// TIA Portal V19 export
DATA_BLOCK "DB_DP"   // DB85
{ S7_Optimized_Access := 'FALSE' }
// stored: AutoNumber false
   VAR RETAIN
      Anz_DP : Int := 2;   // * Anzahl Dosierpumpen
      Offset : Int := 20;   // * Beginn Daten
      leng_Pos : Int := 20;   // * Länge Daten
      DP_Nr : Int := 0;   // Nummer der aktuell bearbeiteten Pumpe
      Sekunden_Takt : Bool := FALSE;   // merkt sich den Sekundentakt
      Minuten_Takt : Bool := FALSE;   // eine Minute ist um (für einen Umlauf an)
      HandeventTakt : Bool := FALSE;   // zyklischer Abstand Meldung manuelle Zugabe
      res1 : Bool := FALSE;
      res2 : Bool := FALSE;
      res3 : Bool := FALSE;
      res4 : Bool := FALSE;
      res5 : Bool := FALSE;
      AM_Minute : Byte := 16#32;   // Altmerker Minute
      MinCount : Int := 1;   // Minutenzähler (10min)
      CheckPU : Int := 0;   // Kontrollpumpe
      resI : Int := 0;
      resD1 : DWord := 16#0000_0000;
      DP : Array[0..20] of Struct   // * Feldlänge anpassen
         Typ : Byte;   // *VAT 0=Menge Zeit,1=Menge Pulse,2=Handzugabe,5=H2O
         LaZa_Nr : Byte;   // *VAT Ladungszähler-Nr.
         EventTime : Int;   // 0=jede Dosierung sonst Zeit in Minuten
         Rest_EventTime : Int;   // Restzeit bis nächstes Event
         DP_Start : Bool;   // Start Dosierpumpe (auch extern 1 Autowert)
         DP_OFF : Bool;   // ext.Abschaltg. zB.Motorschutz oä.
         DP_Hand : Bool;   // Start eine Handzugabe
         DP_Strg : Bool;   // Störung Dosierpumpe
         DP_Imp : Bool;   // externer Zählimpuls
         DP_Niv : Bool;   // Niveau max erreicht
         DP_IN6 : Bool;
         DP_IN7 : Bool;
         DP_IN8 : Bool;
         Dosi_akt : Bool;   // Nachdosierung aktiv
         AM_Dosi : Bool;   // Altmerker Dosierung
         Meldung : Bool;   // Dosierung melden
         AM_Strg : Bool;   // Altmerker Störung
         DP_ext_Imp : Bool;   // Pumpe wird extern betrieben (Impuls wird als Eingang geliefert)
         res4 : Bool;
         AM_DP_Start : Bool;   // Merker DP Start
         RestZeit : Int;   // Restzeit Zähler Dosierimpuls/Pausenzeit
         DosMenge_Auto : Real;   // Dosiermenge Automatik
         DosMenge_Hand : Real;   // Dosiermenge Handzugabe
         ZeitBasis : Byte;   // Zeitbasis für Kalibrierung 0=s 1=min 2=h
         Korr_Einheit : Byte;   // ggf.Korrektur der Einheit
      END_STRUCT;
   END_VAR
BEGIN
   DP[0..20].Typ := 16#00;
   DP[0..20].LaZa_Nr := 16#00;
   DP[0..20].EventTime := 0;
   DP[0..7].Rest_EventTime := 1;
   DP[8..20].Rest_EventTime := 0;
   DP[0..20].DP_Start := FALSE;
   DP[0..20].DP_OFF := FALSE;
   DP[0..20].DP_Hand := FALSE;
   DP[0..20].DP_Strg := FALSE;
   DP[0..20].DP_Imp := FALSE;
   DP[0..20].DP_Niv := FALSE;
   DP[0..20].DP_IN6 := FALSE;
   DP[0..20].DP_IN7 := FALSE;
   DP[0..20].DP_IN8 := FALSE;
   DP[0..20].Dosi_akt := FALSE;
   DP[0..20].AM_Dosi := FALSE;
   DP[0..7].Meldung := TRUE;
   DP[8..20].Meldung := FALSE;
   DP[0..20].AM_Strg := FALSE;
   DP[0..20].DP_ext_Imp := FALSE;
   DP[0..20].res4 := FALSE;
   DP[0..20].AM_DP_Start := FALSE;
   DP[0..20].RestZeit := 0;
   DP[0..20].DosMenge_Auto := 0.0;
   DP[0..20].DosMenge_Hand := 0.0;
   DP[0..20].ZeitBasis := 16#00;
   DP[0..20].Korr_Einheit := 16#00;
END_DATA_BLOCK
